VAR_GLOBAL
	// TIXEL
	{attribute 'TcLinkTo' := '.bLimitForwardEnable:=TIIB[TIXELX-EL7041]^STM Status^Status^Digital input 1;
                              .bLimitBackwardEnable:=TIIB[TIXELX-EL7041]^STM Status^Status^Digital input 2'}
	{attribute 'pytmc' := '
		pv: TMO:LAMP:MMS:10
	'}
	M10		: DUT_MotionStage := (bPowerSelf:=TRUE,
    nEnableMode:=ENUM_StageEnableMode.DURING_MOTION,
    nHomingMode := ENUM_EpicsHomeCmd.ABSOLUTE_SET); // TIXEL X
	
	{attribute 'TcLinkTo' := '.bLimitForwardEnable:=TIIB[TIXELY-EL7041]^STM Status^Status^Digital input 1;
                              .bLimitBackwardEnable:=TIIB[TIXELY-EL7041]^STM Status^Status^Digital input 2'}
	{attribute 'pytmc' := '
		pv: TMO:LAMP:MMS:11
	'}
	M11		: DUT_MotionStage := (bPowerSelf:=TRUE,
    nEnableMode:=ENUM_StageEnableMode.DURING_MOTION,
    nHomingMode := ENUM_EpicsHomeCmd.ABSOLUTE_SET); // TIXEL Y

	{attribute 'TcLinkTo' := '.bLimitForwardEnable:=TIIB[TIXELZ-EL7041]^STM Status^Status^Digital input 1;
                              .bLimitBackwardEnable:=TIIB[TIXELZ-EL7041]^STM Status^Status^Digital input 2'}
	{attribute 'pytmc' := '
		pv: TMO:LAMP:MMS:12
	'}
	M12		: DUT_MotionStage := (bPowerSelf:=TRUE,
    nEnableMode:=ENUM_StageEnableMode.DURING_MOTION,
    nHomingMode := ENUM_EpicsHomeCmd.ABSOLUTE_SET); // TIXEL Z
END_VAR

(* stored: Version 1.1.0.1, ProductVersion 3.1.4022.18
   GVL TIXEL: Id {f1d9ca19-916e-4e8b-b201-c752b93acce4} *)
